// TIA Portal project "memo gra" (V16)

(* hardware
DEVICE "S7-1200 station_1"  S7-1200 Station
   slot 0: "Rack_0"  S7-1200 Rack  Rack  V1.0
   slot 1: "PLC_1"  CPU 1215C DC/DC/DC  6ES7 215-1AG40-0XB0  V4.4
DEVICE "PC-System_1"  SIMATIC PC station
   slot 0: "SIMATIC PC station"  Rail  SIMATIC PC-Station  V1.0
      slot 125: "Stationmanager"  Station_Manager  V6.0.4
   slot 1: "IE general_1"  IE General  IE_CP  V8.2.0
   slot 2: "HMI_RT_1"  WinCC RT Advanced  6AV2 104-0xxxx-xxxx  16.0.0.0
      slot 33792: "Computer interface"  Host interface
*)

// ===== PLC "PLC_1"  CPU 1215C DC/DC/DC =====

VAR_GLOBAL   // PLC tag table "Default tag table"
   "System_Byte" AT %MB1 : Byte;
   "FirstScan" AT %M1.0 : Bool;
   "DiagStatusUpdate" AT %M1.1 : Bool;
   "AlwaysTRUE" AT %M1.2 : Bool;
   "AlwaysFALSE" AT %M1.3 : Bool;
   "Clock_Byte" AT %MB0 : Byte;
   "Clock_10Hz" AT %M0.0 : Bool;
   "Clock_5Hz" AT %M0.1 : Bool;
   "Clock_2.5Hz" AT %M0.2 : Bool;
   "Clock_2Hz" AT %M0.3 : Bool;
   "Clock_1.25Hz" AT %M0.4 : Bool;
   "Clock_1Hz" AT %M0.5 : Bool;
   "Clock_0.625Hz" AT %M0.6 : Bool;
   "Clock_0.5Hz" AT %M0.7 : Bool;
   "lifebit" AT %M5.0 : Bool;
   "Tag_1" AT %MW11 : Int;
   "Tag_2" AT %MW12 : Word;
   "Tag_3" AT %M14.0 : Bool;
   "Tag_4" AT %MW4 : Word;
   "wylosuj liczbe" AT %M20.0 : Bool;
   "Tag_6" AT %M100.0 : Bool;
   "asdsda" AT %MW1 : Int;
   "Nowa gra" AT %M15.0 : Bool;
   "Tag_5" AT %M100.1 : Bool;
   "Tag_7" AT %M61.0 : Bool;
   "Tag_8" AT %M16.0 : Bool;
   "Tag_9" AT %M16.1 : Bool;
   "Tag_10" AT %M120.1 : Bool;
   "Tag_11" AT %M45.0 : Bool;
   "Tag_12" AT %M45.1 : Bool;
   "reset limitu" AT %M50.0 : Bool;
   "wlacz timer" AT %M40.0 : Bool;
   "wlacz timer2" AT %M40.1 : Bool;
   "running" AT %M10.5 : Bool;
   "win" AT %M10.6 : Bool;
   "Tag_13" AT %M65.0 : Bool;
   "Tag_14" AT %M65.1 : Bool;
   "Tag_15" AT %M65.2 : Bool;
   "Tag_16" AT %M65.3 : Bool;
   "Tag_17" AT %M65.4 : Bool;
   "Tag_18" AT %M65.5 : Bool;
   "Tag_19" AT %M65.6 : Bool;
   "Tag_20" AT %M65.7 : Bool;
   "Tag_21" AT %M66.0 : Bool;
   "Tag_22" AT %M66.1 : Bool;
   "Tag_23" AT %M66.2 : Bool;
   "Tag_24" AT %M66.3 : Bool;
   "Tag_25" AT %M66.4 : Bool;
   "Tag_26" AT %M66.5 : Bool;
   "Tag_27" AT %M66.6 : Bool;
   "Tag_28" AT %M66.7 : Bool;
END_VAR

DATA_BLOCK "Data_block_1"   // DB1
{ S7_Optimized_Access := 'TRUE' }
VERSION : 0.1
   VAR
      czas : DTL;
      czas2 : Time_Of_Day;
      "czas w udint" : UDInt;
      "tile array hidden" : Array[1..16] of Int;
      "tile array" : Array[1..16] of Int;
      "zgadniete pola" : Array[1..16] of Int;
      "wylosowana liczba" : Int;
      "wylosowane liczby" : Array[1..16] of Int;
      "tablica wypelniona" : Bool;
      "ilosc ruchow" : Int;
      "detekcja klikniec" : Array[1..16] of Bool;
      "detekcja klikniec2" : Array[1..16] of Bool;
      "limit odkrywania pol" : Int;
      "koniec blednego ruchu" : Bool;
      "koniec dobrego ruchu" : Bool;
      "tryb porownania" : Bool;
      wartosc1 : Int;
      wartosc2 : Int;
      "wartosc1 idx" : Int;
      "wartosc2 idx" : Int;
      bul1 : Bool;
      bul2 : Bool;
   END_VAR
BEGIN
END_DATA_BLOCK

// folder: System blocks/Program resources

DATA_BLOCK "IEC_Counter_0_DB"   // DB2
{ S7_Optimized_Access := 'TRUE' }
AUTHOR : Simatic
FAMILY : IEC
NAME : CNTR
VERSION : 1.0
// stored: InstanceOfName IEC_COUNTER
"IEC_COUNTER"
BEGIN
END_DATA_BLOCK

DATA_BLOCK "IEC_Timer_0_DB_2"   // DB4
{ S7_Optimized_Access := 'TRUE' }
AUTHOR : Simatic
FAMILY : IEC
NAME : IEC_TMR
VERSION : 1.0
// stored: InstanceOfName IEC_TIMER
"IEC_TIMER"
BEGIN
END_DATA_BLOCK

DATA_BLOCK "IEC_Timer_0_DB"   // DB5
{ S7_Optimized_Access := 'TRUE' }
AUTHOR : Simatic
FAMILY : IEC
NAME : IEC_TMR
VERSION : 1.0
// stored: InstanceOfName IEC_TIMER
"IEC_TIMER"
BEGIN
END_DATA_BLOCK

// folder: (top level)

FUNCTION "gra" : Void   // FC1, SCL
{ S7_Optimized_Access := 'TRUE' }
VERSION : 0.1
   VAR_TEMP
      qwe : Int;
      jajo : Int;
   END_VAR
BEGIN
   "reset limitu" := FALSE;

   IF "Data_block_1"."limit odkrywania pol" <= 2 & "Tag_11" THEN
       FOR #qwe := 1 TO 16 DO
           IF "Data_block_1"."detekcja klikniec2"[#qwe] = TRUE & "Data_block_1".wartosc1 = 0 THEN

               EXIT;
               ;
           END_IF;
           ;
       END_FOR;

       FOR #qwe := 1 TO 16 DO
           IF "Data_block_1"."detekcja klikniec2"[#qwe] = TRUE THEN
               "Data_block_1"."tile array"[#qwe] := "Data_block_1"."tile array hidden"[#qwe];
               IF "Data_block_1".wartosc1 = 0 THEN
                   "Data_block_1".wartosc1 := "Data_block_1"."tile array"[#qwe];
                   "Data_block_1"."wartosc1 idx" := #qwe;
                   ;
               END_IF;
               "Data_block_1".wartosc2 := "Data_block_1"."tile array"[#qwe];
               "Data_block_1"."wartosc2 idx" := #qwe;
               ;
           END_IF;
           ;
       END_FOR;
       ;
   END_IF;

   "R_TRIG_DB"(CLK:="Data_block_1"."limit odkrywania pol" = 2,
               Q=>"Data_block_1".bul1);
   IF "Data_block_1".bul1 = TRUE THEN
       "Data_block_1"."ilosc ruchow" += 1;

       IF "Data_block_1".wartosc1 = "Data_block_1".wartosc2 THEN
           "wlacz timer2" := TRUE;
           ;
       ELSE
           "wlacz timer" := TRUE;
           ;
       END_IF;
       ;
   END_IF;

   IF "Data_block_1"."koniec blednego ruchu" THEN
       "wlacz timer" := false;
       "Data_block_1"."tile array"["Data_block_1"."wartosc1 idx"] := 0;
       "Data_block_1"."tile array"["Data_block_1"."wartosc2 idx"] := 0;
       "Data_block_1".wartosc1 := 0;
       "Data_block_1".wartosc2 := 0;
       "Data_block_1"."wartosc1 idx" := 0;
       "Data_block_1"."wartosc2 idx" := 0;
       "reset limitu" := TRUE;
       ;
   END_IF;

   IF "Data_block_1"."koniec dobrego ruchu" THEN
       "wlacz timer2" := FALSE;
       "Data_block_1".wartosc1 := 0;
       "Data_block_1".wartosc2 := 0;
       "Data_block_1"."wartosc1 idx" := 0;
       "Data_block_1"."wartosc2 idx" := 0;
       "reset limitu" := TRUE;
       ;
   END_IF;


   FOR #jajo := 1 TO 16 DO
       IF "Data_block_1"."tile array"[#jajo] = 0 THEN
           EXIT;
           ;
       END_IF;
       IF #jajo = 16 THEN
           "win" := TRUE;
           ;
       END_IF;
       ;
   END_FOR;

   FOR #qwe := 1 TO 16 DO
       "Data_block_1"."detekcja klikniec2"[#qwe] := FALSE;
       ;
   END_FOR;
END_FUNCTION

FUNCTION "timer" : Void   // FC2, LAD
{ S7_Optimized_Access := 'TRUE' }
VERSION : 0.1
BEGIN

REGION Network 1
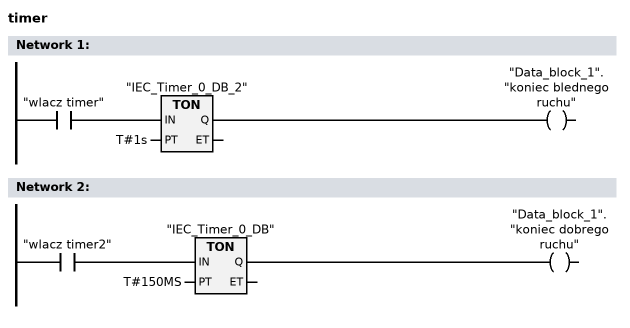
   "IEC_Timer_0_DB_2".TON(IN := "wlacz timer", PT := T#1s);
   "Data_block_1"."koniec blednego ruchu" := "IEC_Timer_0_DB_2".Q;
END_REGION

REGION Network 2
   "IEC_Timer_0_DB".TON(IN := "wlacz timer2", PT := T#150MS);
   "Data_block_1"."koniec dobrego ruchu" := "IEC_Timer_0_DB".Q;
END_REGION
END_FUNCTION

FUNCTION "wypelnianie planszy" : Void   // FC3, SCL
{ S7_Optimized_Access := 'TRUE' }
VERSION : 0.1
   VAR_TEMP
      asd : Int;
      asd2 : Int;
      asd3 : Int;
      "wylosowano nowa" : Bool;
      asd4 : Int;
      asd5 : Int;
   END_VAR
BEGIN
   #asd2 := 1;

   "wylosuj liczbe" := FALSE;

   FOR #asd := 1 TO 8 DO
       //sprawdza czy wylosowana liczba juz sie pojawila
       #"wylosowano nowa" := FALSE;
       WHILE #"wylosowano nowa" <> TRUE DO
           "Tag_1" := RD_LOC_T("Data_block_1".czas);
           "Data_block_1".czas2 := DTL_TO_TOD("Data_block_1".czas);
           "Data_block_1"."czas w udint" := TOD_TO_UDINT("Data_block_1".czas2);
           "Data_block_1"."wylosowana liczba" := "Data_block_1"."czas w udint" MOD 16;
           "Data_block_1"."wylosowana liczba" += 1;

           #"wylosowano nowa" := TRUE;
           FOR #asd3 := 1 TO 16 DO
               IF "Data_block_1"."wylosowana liczba" = "Data_block_1"."wylosowane liczby"[#asd3] THEN
                   #"wylosowano nowa" := FALSE;
                   EXIT;
                   ;
               END_IF;
               ;
           END_FOR;
           ;
       END_WHILE;


       "Data_block_1"."tile array hidden"["Data_block_1"."wylosowana liczba"] := #asd;
       "Data_block_1"."wylosowane liczby"[#asd2] := "Data_block_1"."wylosowana liczba";

       #asd2 += 1;


       IF #asd2 = 16 THEN
           FOR #asd4 := 1 TO 16 DO
               IF "Data_block_1"."tile array hidden"[#asd4] = 0 THEN
                   "Data_block_1"."tile array hidden"[#asd4] := #asd;
                   EXIT;
                   ;
               END_IF;
               ;
           END_FOR;
           EXIT;
           ;
       END_IF;

       //sprawdza czy wylosowana liczba juz sie pojawila
       #"wylosowano nowa" := FALSE;
       WHILE #"wylosowano nowa" <> TRUE DO
           "Tag_1" := RD_LOC_T("Data_block_1".czas);
           "Data_block_1".czas2 := DTL_TO_TOD("Data_block_1".czas);
           "Data_block_1"."czas w udint" := TOD_TO_UDINT("Data_block_1".czas2);
           "Data_block_1"."wylosowana liczba" := "Data_block_1"."czas w udint" MOD 15;
           "Data_block_1"."wylosowana liczba" += 1;

           #"wylosowano nowa" := TRUE;
           FOR #asd3 := 1 TO 16 DO
               IF "Data_block_1"."wylosowana liczba" = "Data_block_1"."wylosowane liczby"[#asd3] THEN
                   #"wylosowano nowa" := FALSE;
                   EXIT;
                   ;
               END_IF;
               ;
           END_FOR;
           ;
       END_WHILE;

       "Data_block_1"."tile array hidden"["Data_block_1"."wylosowana liczba"] := #asd;
       "Data_block_1"."wylosowane liczby"[#asd2] := "Data_block_1"."wylosowana liczba";

       #asd2 += 1;
       ;
   END_FOR;

   "Data_block_1"."tablica wypelniona" := true;
END_FUNCTION

FUNCTION "obxluga przyciskow" : Void   // FC4, LAD
{ S7_Optimized_Access := 'TRUE' }
VERSION : 0.1
   VAR_TEMP   // added for the SCL form of the ladder/FBD networks
      _w1 : Bool;
      _w2 : Bool;
      _w3 : Bool;
      _w4 : Bool;
      _w5 : Bool;
      _w6 : Bool;
      _w7 : Bool;
      _w8 : Bool;
      _w9 : Bool;
      _w10 : Bool;
      _w11 : Bool;
      _w12 : Bool;
      _w13 : Bool;
      _w14 : Bool;
      _w15 : Bool;
      _w16 : Bool;
      _w17 : Bool;
      _w18 : Bool;
   END_VAR
BEGIN

REGION Network 1
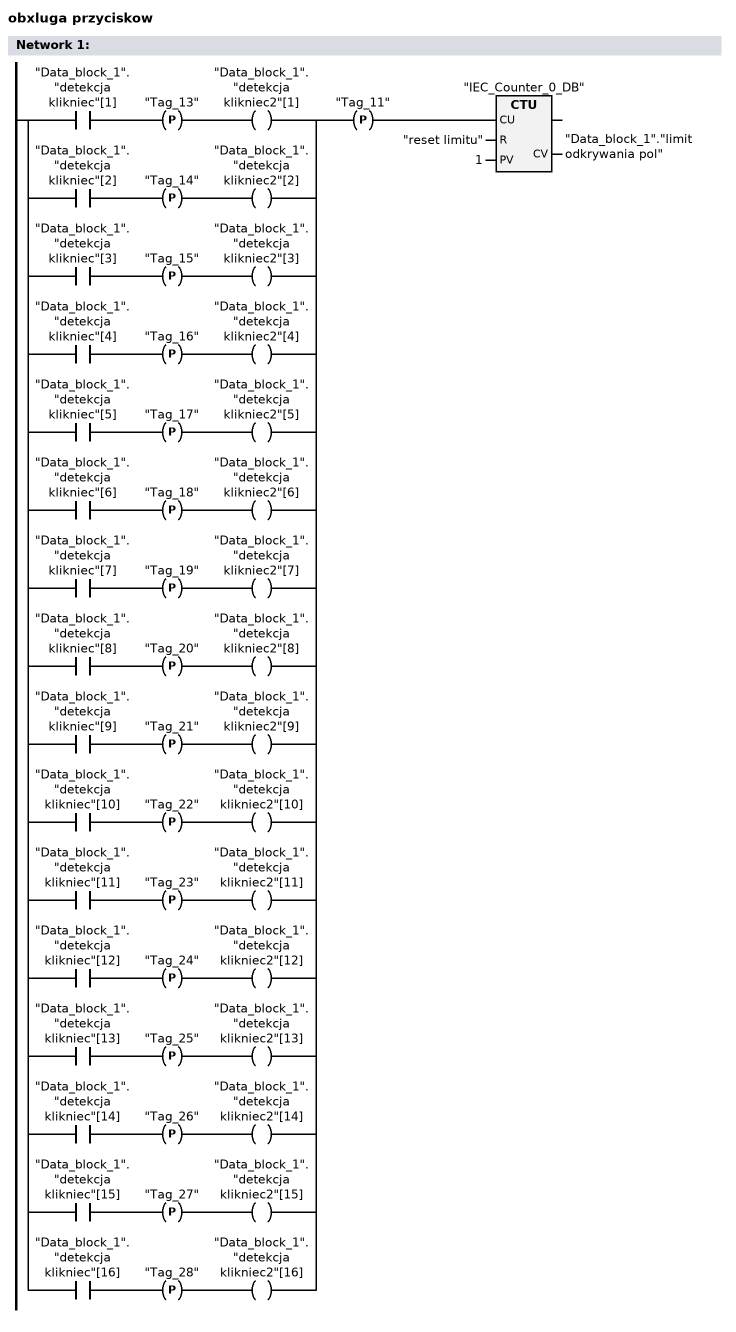
   #_w1 := "Data_block_1"."detekcja klikniec"[1] AND NOT "Tag_13";   // rising edge
   "Tag_13" := "Data_block_1"."detekcja klikniec"[1];
   "Data_block_1"."detekcja klikniec2"[1] := #_w1;
   #_w2 := "Data_block_1"."detekcja klikniec"[2] AND NOT "Tag_14";   // rising edge
   "Tag_14" := "Data_block_1"."detekcja klikniec"[2];
   "Data_block_1"."detekcja klikniec2"[2] := #_w2;
   #_w3 := "Data_block_1"."detekcja klikniec"[3] AND NOT "Tag_15";   // rising edge
   "Tag_15" := "Data_block_1"."detekcja klikniec"[3];
   "Data_block_1"."detekcja klikniec2"[3] := #_w3;
   #_w4 := "Data_block_1"."detekcja klikniec"[4] AND NOT "Tag_16";   // rising edge
   "Tag_16" := "Data_block_1"."detekcja klikniec"[4];
   "Data_block_1"."detekcja klikniec2"[4] := #_w4;
   #_w5 := "Data_block_1"."detekcja klikniec"[5] AND NOT "Tag_17";   // rising edge
   "Tag_17" := "Data_block_1"."detekcja klikniec"[5];
   "Data_block_1"."detekcja klikniec2"[5] := #_w5;
   #_w6 := "Data_block_1"."detekcja klikniec"[6] AND NOT "Tag_18";   // rising edge
   "Tag_18" := "Data_block_1"."detekcja klikniec"[6];
   "Data_block_1"."detekcja klikniec2"[6] := #_w6;
   #_w7 := "Data_block_1"."detekcja klikniec"[7] AND NOT "Tag_19";   // rising edge
   "Tag_19" := "Data_block_1"."detekcja klikniec"[7];
   "Data_block_1"."detekcja klikniec2"[7] := #_w7;
   #_w8 := "Data_block_1"."detekcja klikniec"[8] AND NOT "Tag_20";   // rising edge
   "Tag_20" := "Data_block_1"."detekcja klikniec"[8];
   "Data_block_1"."detekcja klikniec2"[8] := #_w8;
   #_w9 := "Data_block_1"."detekcja klikniec"[9] AND NOT "Tag_21";   // rising edge
   "Tag_21" := "Data_block_1"."detekcja klikniec"[9];
   "Data_block_1"."detekcja klikniec2"[9] := #_w9;
   #_w10 := "Data_block_1"."detekcja klikniec"[10] AND NOT "Tag_22";   // rising edge
   "Tag_22" := "Data_block_1"."detekcja klikniec"[10];
   "Data_block_1"."detekcja klikniec2"[10] := #_w10;
   #_w11 := "Data_block_1"."detekcja klikniec"[11] AND NOT "Tag_23";   // rising edge
   "Tag_23" := "Data_block_1"."detekcja klikniec"[11];
   "Data_block_1"."detekcja klikniec2"[11] := #_w11;
   #_w12 := "Data_block_1"."detekcja klikniec"[12] AND NOT "Tag_24";   // rising edge
   "Tag_24" := "Data_block_1"."detekcja klikniec"[12];
   "Data_block_1"."detekcja klikniec2"[12] := #_w12;
   #_w13 := "Data_block_1"."detekcja klikniec"[13] AND NOT "Tag_25";   // rising edge
   "Tag_25" := "Data_block_1"."detekcja klikniec"[13];
   "Data_block_1"."detekcja klikniec2"[13] := #_w13;
   #_w14 := "Data_block_1"."detekcja klikniec"[14] AND NOT "Tag_26";   // rising edge
   "Tag_26" := "Data_block_1"."detekcja klikniec"[14];
   "Data_block_1"."detekcja klikniec2"[14] := #_w14;
   #_w15 := "Data_block_1"."detekcja klikniec"[15] AND NOT "Tag_27";   // rising edge
   "Tag_27" := "Data_block_1"."detekcja klikniec"[15];
   "Data_block_1"."detekcja klikniec2"[15] := #_w15;
   #_w16 := "Data_block_1"."detekcja klikniec"[16] AND NOT "Tag_28";   // rising edge
   "Tag_28" := "Data_block_1"."detekcja klikniec"[16];
   "Data_block_1"."detekcja klikniec2"[16] := #_w16;
   #_w17 := #_w1 OR #_w2 OR #_w3 OR #_w4 OR #_w5 OR #_w6 OR #_w7 OR #_w8 OR #_w9 OR #_w10 OR #_w11 OR #_w12 OR #_w13 OR #_w14 OR #_w15 OR #_w16;
   #_w18 := #_w17 AND NOT "Tag_11";   // rising edge
   "Tag_11" := #_w17;
   "IEC_Counter_0_DB".CTU(CU := #_w18,
                          R := "reset limitu",
                          PV := 1,
                          CV => "Data_block_1"."limit odkrywania pol");
END_REGION
END_FUNCTION

FUNCTION "czyszczenie pamieci" : Void   // FC5, SCL
{ S7_Optimized_Access := 'TRUE' }
VERSION : 0.1
   VAR_TEMP
      asd5 : Int;
   END_VAR
BEGIN
   FOR #asd5 := 1 TO 16 DO
       "Data_block_1"."tile array"[#asd5] := 0;
       "Data_block_1"."tile array hidden"[#asd5] := 0;
       "Data_block_1"."wylosowane liczby"[#asd5] := 0;
       "Data_block_1"."detekcja klikniec"[#asd5] := 0;
       ;
   END_FOR;

   "Data_block_1"."tablica wypelniona" := FALSE;
   "Data_block_1"."ilosc ruchow" := 0;
   "Data_block_1".wartosc1 := 0;
   "Data_block_1".wartosc2 := 0;
   "Data_block_1"."wartosc1 idx" := 0;
   "Data_block_1"."wartosc2 idx" := 0;

   "Data_block_1"."tryb porownania" := FALSE;
   "win" := FALSE;
END_FUNCTION

ORGANIZATION_BLOCK "Main"   // OB1, LAD, ProgramCycle
TITLE = "Main Program Sweep (Cycle)"
{ S7_Optimized_Access := 'TRUE' }
VERSION : 0.1
   VAR_INPUT
      Initial_Call : Bool;   // Initial call of this OB
      Remanence : Bool;   // =True, if remanent data are available
   END_VAR
   VAR_TEMP   // added for the SCL form of the ladder/FBD networks
      _w1 : Bool;
      _w2 : Bool;
   END_VAR
BEGIN

REGION Network 1
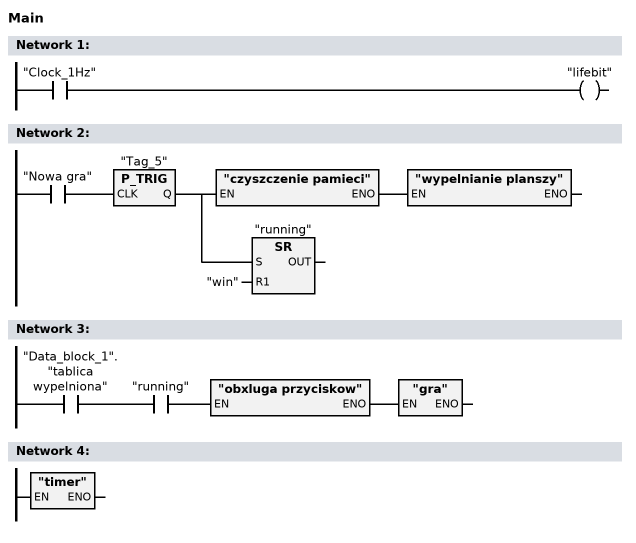
   RUNG wire#powerrail
      Contact( "Clock_1Hz" )
      Coil( "lifebit" )
   END_RUNG
   // the same network as SCL:
   "lifebit" := "Clock_1Hz";
END_REGION

REGION Network 2
   RUNG wire#powerrail
      Contact( "Nowa gra" )
      P_Trig( "Tag_5" )
      wire#w1
      "czyszczenie pamieci"()
      "wypelnianie planszy"()
   END_RUNG
   RUNG wire#w1
      S_SR(operand := "running", r1 := "win")
   END_RUNG
   // the same network as SCL:
   #_w1 := "Nowa gra" AND NOT "Tag_5";   // rising edge
   "Tag_5" := "Nowa gra";
   "czyszczenie pamieci"(EN := #_w1, ENO => #_w2);
   IF #_w2 THEN "wypelnianie planszy"(); END_IF;
   IF #_w1 THEN
       "running" := TRUE;   // SR flip-flop
   END_IF;
   IF "win" THEN "running" := FALSE; END_IF;
END_REGION

REGION Network 3
   RUNG wire#powerrail
      Contact( "Data_block_1"."tablica wypelniona" )
      Contact( "running" )
      "obxluga przyciskow"()
      "gra"()
   END_RUNG
   // the same network as SCL:
   "obxluga przyciskow"(EN := "Data_block_1"."tablica wypelniona" AND "running", ENO => #_w1);
   IF #_w1 THEN "gra"(); END_IF;
END_REGION

REGION Network 4
   RUNG wire#powerrail
      "timer"()
   END_RUNG
   // the same network as SCL:
   "timer"();
END_REGION
END_ORGANIZATION_BLOCK

(* ===== HMI "HMI_RT_1" =====
system functions are stored by id; their names below are inferred from use
connection "HMI_Connection_1": ETHERNET, S7_1200_OMS

HMI tags "Default tag table"
   "lifebit" : Bool = PLC lifebit AT %M5.0, 100 ms
   "wylosuj liczbe" : Bool = PLC "wylosuj liczbe" AT %M20.0, 100 ms
   "Data_block_1_wylosowana liczba" : Int = PLC Data_block_1."wylosowana liczba", 100 ms
   "Data_block_1_tile array{1}" : Int = PLC Data_block_1."tile array"[1], 100 ms
   "Data_block_1_tile array{2}" : Int = PLC Data_block_1."tile array"[2], 100 ms
   "Data_block_1_tile array{3}" : Int = PLC Data_block_1."tile array"[3], 100 ms
   "Data_block_1_tile array{4}" : Int = PLC Data_block_1."tile array"[4], 100 ms
   "Data_block_1_tile array{5}" : Int = PLC Data_block_1."tile array"[5], 100 ms
   "Data_block_1_tile array{6}" : Int = PLC Data_block_1."tile array"[6], 100 ms
   "Data_block_1_tile array{7}" : Int = PLC Data_block_1."tile array"[7], 100 ms
   "Data_block_1_tile array{8}" : Int = PLC Data_block_1."tile array"[8], 100 ms
   "Data_block_1_tile array{9}" : Int = PLC Data_block_1."tile array"[9], 100 ms
   "Data_block_1_tile array{10}" : Int = PLC Data_block_1."tile array"[10], 100 ms
   "Data_block_1_tile array{11}" : Int = PLC Data_block_1."tile array"[11], 100 ms
   "Data_block_1_tile array{12}" : Int = PLC Data_block_1."tile array"[12], 100 ms
   "Data_block_1_tile array{13}" : Int = PLC Data_block_1."tile array"[13], 100 ms
   "Data_block_1_tile array{14}" : Int = PLC Data_block_1."tile array"[14], 100 ms
   "Data_block_1_tile array{15}" : Int = PLC Data_block_1."tile array"[15], 100 ms
   "Data_block_1_tile array{16}" : Int = PLC Data_block_1."tile array"[16], 100 ms
   "Nowa gra" : Bool = PLC "Nowa gra" AT %M15.0, 100 ms
   "Data_block_1_detekcja klikniec{1}" : Bool = PLC Data_block_1."detekcja klikniec"[1], 1 s
   "Data_block_1_detekcja klikniec{2}" : Bool = PLC Data_block_1."detekcja klikniec"[2], 1 s
   "Data_block_1_detekcja klikniec{3}" : Bool = PLC Data_block_1."detekcja klikniec"[3], 1 s
   "Data_block_1_detekcja klikniec{4}" : Bool = PLC Data_block_1."detekcja klikniec"[4], 1 s
   "Data_block_1_detekcja klikniec{5}" : Bool = PLC Data_block_1."detekcja klikniec"[5], 1 s
   "Data_block_1_detekcja klikniec{6}" : Bool = PLC Data_block_1."detekcja klikniec"[6], 1 s
   "Data_block_1_detekcja klikniec{7}" : Bool = PLC Data_block_1."detekcja klikniec"[7], 1 s
   "Data_block_1_detekcja klikniec{8}" : Bool = PLC Data_block_1."detekcja klikniec"[8], 1 s
   "Data_block_1_detekcja klikniec{9}" : Bool = PLC Data_block_1."detekcja klikniec"[9], 1 s
   "Data_block_1_detekcja klikniec{10}" : Bool = PLC Data_block_1."detekcja klikniec"[10], 1 s
   "Data_block_1_detekcja klikniec{11}" : Bool = PLC Data_block_1."detekcja klikniec"[11], 1 s
   "Data_block_1_detekcja klikniec{12}" : Bool = PLC Data_block_1."detekcja klikniec"[12], 1 s
   "Data_block_1_detekcja klikniec{13}" : Bool = PLC Data_block_1."detekcja klikniec"[13], 1 s
   "Data_block_1_detekcja klikniec{14}" : Bool = PLC Data_block_1."detekcja klikniec"[14], 1 s
   "Data_block_1_detekcja klikniec{15}" : Bool = PLC Data_block_1."detekcja klikniec"[15], 1 s
   "Data_block_1_detekcja klikniec{16}" : Bool = PLC Data_block_1."detekcja klikniec"[16], 1 s
   "Data_block_1_ilosc ruchow" : Int = PLC Data_block_1."ilosc ruchow", 1 s
   "reset limitu" : Bool = PLC "reset limitu" AT %M50.0, 1 s
   "win" : Bool = PLC win AT %M10.6, 1 s

screen "Screen_1" 1024x768
   Circle "Circle_1" at 0,0 size 48x48
      Appearance <- "lifebit"
   DateTimeField "Date/time field_1" at 804,8 size 212x31
   Button "Button_2" at 59,185 size 96x32; TextOff 'Nowa Gra'
      on Press: function_b14e0dd5("Nowa gra", 0); function_b14e0dd5("reset limitu", 0)
   Group "Group" at 309,182 size 100x100; FormatPattern 9999999
   Group "Group_1" at 409,182 size 100x100; FormatPattern 9999999
   Group "Group_2" at 509,182 size 100x100; FormatPattern 9999999
   Group "Group_3" at 609,182 size 100x100; FormatPattern 9999999
   Group "Group_4" at 309,282 size 100x100; FormatPattern 9999999
   Group "Group_5" at 409,282 size 100x100; FormatPattern 9999999
   Group "Group_6" at 509,282 size 100x100; FormatPattern 9999999
   Group "Group_7" at 609,282 size 100x100; FormatPattern 9999999
   Group "Group_8" at 309,382 size 100x100; FormatPattern 9999999
   Group "Group_9" at 409,382 size 100x100; FormatPattern 9999999
   Group "Group_10" at 509,382 size 100x100; FormatPattern 9999999
   Group "Group_11" at 609,382 size 100x100; FormatPattern 9999999
   Group "Group_12" at 309,482 size 100x100; FormatPattern 9999999
   Group "Group_13" at 409,482 size 100x100; FormatPattern 9999999
   Group "Group_14" at 509,482 size 100x100; FormatPattern 9999999
   Group "Group_15" at 609,482 size 100x100; FormatPattern 9999999
   IOField "I/O field_1" at 453,63 size 96x32; FormatPattern 99999
      ProcessValue <- "Data_block_1_ilosc ruchow"
   TextField "Text field_1" at 350,68 size 101x22; Text 'Ilość ruchów'
   Group "Group_16" at 453,112 size 96x48
   IOField "I/O field_2" at 309,182 size 100x100; FormatPattern 99
      ProcessValue <- "Data_block_1_tile array{1}"
   Button "Button_1" at 309,182 size 100x100; TextOff '1'
      on Press: function_b14e0dd5("Data_block_1_detekcja klikniec{1}", 0)
   IOField "I/O field_3" at 409,182 size 100x100; FormatPattern 99
      ProcessValue <- "Data_block_1_tile array{2}"
   Button "Button_3" at 409,182 size 100x100; TextOff 'Text'
      on Press: function_b14e0dd5("Data_block_1_detekcja klikniec{2}", 0)
   IOField "I/O field_4" at 509,182 size 100x100; FormatPattern 99
      ProcessValue <- "Data_block_1_tile array{3}"
   Button "Button_4" at 509,182 size 100x100; TextOff 'Text'
      on Press: function_b14e0dd5("Data_block_1_detekcja klikniec{3}", 0)
   IOField "I/O field_5" at 609,182 size 100x100; FormatPattern 99
      ProcessValue <- "Data_block_1_tile array{4}"
   Button "Button_5" at 609,182 size 100x100; TextOff 'Text'
      on Press: function_b14e0dd5("Data_block_1_detekcja klikniec{4}", 0)
   IOField "I/O field_6" at 309,282 size 100x100; FormatPattern 99
      ProcessValue <- "Data_block_1_tile array{5}"
   Button "Button_6" at 309,282 size 100x100; TextOff 'Text'
      on Press: function_b14e0dd5("Data_block_1_detekcja klikniec{5}", 0)
   IOField "I/O field_7" at 409,282 size 100x100; FormatPattern 99
      ProcessValue <- "Data_block_1_tile array{6}"
   Button "Button_7" at 409,282 size 100x100; TextOff 'Text'
      on Press: function_b14e0dd5("Data_block_1_detekcja klikniec{6}", 0)
   IOField "I/O field_8" at 509,282 size 100x100; FormatPattern 99
      ProcessValue <- "Data_block_1_tile array{7}"
   Button "Button_8" at 509,282 size 100x100; TextOff 'Text'
      on Press: function_b14e0dd5("Data_block_1_detekcja klikniec{7}", 0)
   IOField "I/O field_9" at 609,282 size 100x100; FormatPattern 99
      ProcessValue <- "Data_block_1_tile array{8}"
   Button "Button_9" at 609,282 size 100x100; TextOff 'Text'
      on Press: function_b14e0dd5("Data_block_1_detekcja klikniec{8}", 0)
   IOField "I/O field_10" at 309,382 size 100x100; FormatPattern 99
      ProcessValue <- "Data_block_1_tile array{9}"
   Button "Button_10" at 309,382 size 100x100; TextOff 'Text'
      on Press: function_b14e0dd5("Data_block_1_detekcja klikniec{9}", 0)
   IOField "I/O field_11" at 409,382 size 100x100; FormatPattern 99
      ProcessValue <- "Data_block_1_tile array{10}"
   Button "Button_11" at 409,382 size 100x100; TextOff 'Text'
      on Press: function_b14e0dd5("Data_block_1_detekcja klikniec{10}", 0)
   IOField "I/O field_12" at 509,382 size 100x100; FormatPattern 99
      ProcessValue <- "Data_block_1_tile array{11}"
   Button "Button_12" at 509,382 size 100x100; TextOff 'Text'
      on Press: function_b14e0dd5("Data_block_1_detekcja klikniec{11}", 0)
   IOField "I/O field_13" at 609,382 size 100x100; FormatPattern 99
      ProcessValue <- "Data_block_1_tile array{12}"
   Button "Button_13" at 609,382 size 100x100; TextOff 'Text'
      on Press: function_b14e0dd5("Data_block_1_detekcja klikniec{12}", 0)
   IOField "I/O field_14" at 309,482 size 100x100; FormatPattern 99
      ProcessValue <- "Data_block_1_tile array{13}"
   Button "Button_14" at 309,482 size 100x100; TextOff 'Text'
      on Press: function_b14e0dd5("Data_block_1_detekcja klikniec{13}", 0)
   IOField "I/O field_15" at 409,482 size 100x100; FormatPattern 99
      ProcessValue <- "Data_block_1_tile array{14}"
   Button "Button_15" at 409,482 size 100x100; TextOff 'Text'
      on Press: function_b14e0dd5("Data_block_1_detekcja klikniec{14}", 0)
   IOField "I/O field_16" at 509,482 size 100x100; FormatPattern 99
      ProcessValue <- "Data_block_1_tile array{15}"
   Button "Button_16" at 509,482 size 100x100; TextOff 'Text'
      on Press: function_b14e0dd5("Data_block_1_detekcja klikniec{15}", 0)
   IOField "I/O field_17" at 609,482 size 100x100; FormatPattern 99
      ProcessValue <- "Data_block_1_tile array{16}"
   Button "Button_17" at 609,482 size 100x100; TextOff 'Text'
      on Press: function_b14e0dd5("Data_block_1_detekcja klikniec{16}", 0)
   Rectangle "Rectangle_2" at 453,112 size 96x48
      Visibility <- "win"
   TextField "Text field_2" at 482,128 size 34x22; Text 'Win'
      Visibility <- "win"
*)